// TIA Portal V20 export
FUNCTION_BLOCK "CalledInPreInterpolator"   // FB211, LAD
// stored: Access Published, MemoryReserve 100, Namespace Unit1.Em0, SetENOAutomatically false
BEGIN

REGION Network 1
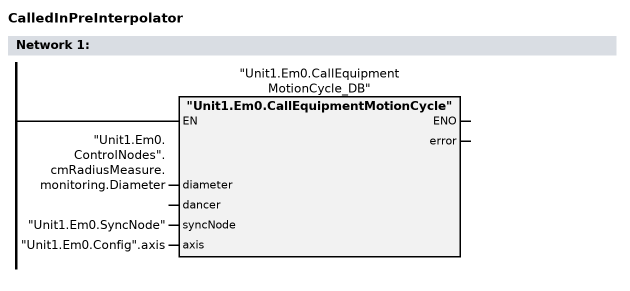
   RUNG wire#powerrail
      "Unit1.Em0.CallEquipmentMotionCycle_DB"(diameter := "Unit1.Em0.ControlNodes".cmRadiusMeasure.monitoring.Diameter, dancer :=, syncNode := "Unit1.Em0.SyncNode", axis := "Unit1.Em0.Config".axis, error =>)
   END_RUNG
   // the same network as SCL:
   "Unit1.Em0.CallEquipmentMotionCycle_DB"(diameter := "Unit1.Em0.ControlNodes".cmRadiusMeasure.monitoring.Diameter,   // "Unit1.Em0.CallEquipmentMotionCycle"
                           syncNode := "Unit1.Em0.SyncNode",
                           axis := "Unit1.Em0.Config".axis);
END_REGION
END_FUNCTION_BLOCK
